Fanuc KAREL source: ke00002.KL

PROGRAM KE00002
%STACKSIZE=65535
%PRIORITY=65535
%NOLOCKGROUP
VAR
S : STRING[80]
I : INTEGER
V : ARRAY[4] OF STRING[80]
K : ARRAY[4] OF STRING[80]
STATUS : INTEGER
BEGIN
S='TEST'
I=1
-- UNRESOLVED_PC line 13 opcodes [3F 22 9D 33 61] marker_code=29
READ_DICT_V(S,I,V,K,STATUS)
END KE00002
